TYPE ST_MotionlinxAI_Controller_Status :
	STRUCT
		Extended   : BOOL;
		Retracted  : BOOL;
		Extending  : BOOL;
		Retracting : BOOL;
	END_STRUCT
END_TYPE

(* stored: Version 1.1.0.1, ProductVersion 3.1.4024.15
   DUT ST_MotionlinxAI_Controller_Status: Id {2441b4da-f342-4f2f-8e84-8a79aa390bb4} *)
